// TIA Portal V16 export
// export: Created 2021-11-12T13:32:03.5567282Z, ExportSetting WithDefaults, DisplayName Totally Integrated Automation Portal, DisplayVersion V16 Update 3, DisplayName TIA Portal Version Control Interface, DisplayVersion V16 Update 2, DisplayName TIA Portal Openness, DisplayVersion V16 Update 3, DisplayName SINAMICS Startdrive Advanced, DisplayVersion V16 Update 5, DisplayName SINAMICS Startdrive G130, G150, S120, S150, SINAMICS MV, S210, DisplayVersion V16 Update 5, DisplayName SINAMICS Startdrive G110M, G120, G120C, G120D, G120P, G115D, DisplayVersion V16 Update 5, DisplayName STEP 7 Professional, DisplayVersion V16 Update 3, DisplayName STEP 7 Safety, DisplayVersion V16, DisplayName WinCC UA Professional, DisplayVersion V16 Update 3
DATA_BLOCK "STATUS_110"   // DB201
{ S7_Optimized_Access := 'TRUE' }
VERSION : 0.1
// stored: AutoNumber true, DBAccessibleFromOPCUA true, IsOnlyStoredInLoadMemory false, IsRetainMemResEnabled false, IsWriteProtectedInAS false, MemoryReserve 100
   VAR
      xxxxx___BinarySensors___xxxxx : Byte;
      GL01_BG01 : Bool;   // Proximitní senzor - Koncák pro referenci
      GL01_BG01R : Bool;   // Proximitní senzor - Zarážka nahoře
      GL01_BG01V : Bool;   // Proximitní senzor - Zarážka dole
      GL01_BG02 : Bool;   // Optický senzor - Přítomnost přířezu v pozici po vykulení
      GM01_BG01R : Bool;   // Indukční senzor - Výtah 1 dole
      GM01_BG01V : Bool;   // Indukční senzor - Výtah 1 nahoře
      GM01_BG02R : Bool;   // Indukční senzor - Výtah 2 dole
      GM01_BG02V : Bool;   // Indukční senzor - Výtah 2 nahoře
      GM01_BG03R : Bool;   // Indukční senzor - Výtah 3 dole
      GM01_BG03V : Bool;   // Indukční senzor - Výtah 3 nahoře
      GM01_BG04R : Bool;   // Indukční senzor - Výtah 4 dole
      GM01_BG04V : Bool;   // Indukční senzor - Výtah 4 nahoře
      GL01_BG03 : Bool;   // Optický senzor - Přířez na řetěze před výtahama
      GM01_BG01 : Bool;   // Optický senzor - Přířez na řetěze výtah 1
      GM01_BG02 : Bool;   // Optický senzor - Přířez na řetěze výtah 2
      GM01_BG03 : Bool;   // Optický senzor - Přířez na řetěze výtah 3
      GM01_BG04 : Bool;   // Optický senzor - Přířez na řetěze výtah 4
      GL01_BG04 : Bool;   // Přířez na řetěze za posledním výtahem
      GL01_BG5 : Bool;   // Enkodér na dopravníku
      xxxxx___BinaryOthers___xxxxx : Byte;
      UH31_FC01 : Bool;   // Servodrive TA01 is OK / Servoměnič TA01 je OK
      UC10_FC21 : Bool;   // 230V Part align OK
      UC12_FC01 : Bool;   // 400V Conveyor OK
      SF01_14 : Bool;   // Conveyor Remote
      SF01_24 : Bool;   // Conveyor Automat
      SF03_14 : Bool;   // Conveyor Start automat
      SF04_12 : Bool;   // Conveyor Stop
      SF05_14 : Bool;   // Conveyor Manual backward
      SF05_24 : Bool;   // Conveyor Manual forward
      SF06_14 : Bool;   // Conveyor lift 1 up
      SF06_24 : Bool;   // Conveyor lift 1 down
      SF07_14 : Bool;   // Conveyor lift 2 up
      SF07_24 : Bool;   // Conveyor lift 2 down
      SF08_14 : Bool;   // Conveyor lift 3 up
      SF08_24 : Bool;   // Conveyor lift 3 down
      SF09_14 : Bool;   // Conveyor lift 4 up
      SF09_24 : Bool;   // Conveyor lift 4 down
      SF10_14 : Bool;   // Conveyor aligning align
      SF10_24 : Bool;   // Conveyor aligning release
      SF11_14 : Bool;   // Conveyor Stopper up
      SF11_24 : Bool;   // Conveyor Stopper down
      xxxxx___Drives___xxxxx : Byte;
      GL01_MA02 : Struct   // Conveyour - motor / Dopravník - motor
         Main : "UDT_Status_main";
         Specific { S7_SetPoint := 'True'} : "UDT_Drive1_Status_specific";
         Error : "UDT_Error01";
      END_STRUCT;
      UC12_TA01 : Struct   // Conveyour - G120 / Dopravník - měnič G120
         Main { S7_SetPoint := 'True'} : "UDT_Status_main";
         Specific { S7_SetPoint := 'True'} : "UDT_SINAMICS_G120_Status_specific";
         Error { S7_SetPoint := 'True'} : "UDT_Error02";
      END_STRUCT;
      GL01_BG05 : Struct   // Conveyour - encoder / Dopravník - enkodér
         Main : "UDT_Status_main";
         Specific : "UDT_MCEncoder_Status_specific";
         Error : "UDT_Error01";
      END_STRUCT;
      UH31_TA01 : Struct   // Servodrive - FESTO / Řízení servomotoru - FESTO
         Main : "UDT_Status_main";
         Specific { S7_SetPoint := 'True'} : "UDT_FESTO_CMMT_Status_specific";
         Error { S7_SetPoint := 'True'} : "UDT_Error02";
      END_STRUCT;
      xxxxx___Others___xxxxx : Byte;
      ConvReadyLoad : Bool;   // Station is ready for material / Stanice je připravena na příjem kusů
      GL01_MA01_HomePos : Bool;   // FESTO servo home position
      PartCounter : Int;   // Number of parts in gripper
      xxxxx___Valves___xxxxx : Byte;
      GL01_MM01 : Struct   // Valve - stopping / Pneumatický válec - Zarážka pro vykulení
         Main : "UDT_Status_main";
         Specific : "UDT_Valve2WB_Status_specific";
         Error : "UDT_Error01";
      END_STRUCT;
      GM01_MM01 : Struct   // Valve - Lift 1 / Pneumatický válec - Zvedání přířezu - Výtah 1
         Main : "UDT_Status_main";
         Specific : "UDT_Valve2WB_Status_specific";
         Error : "UDT_Error01";
      END_STRUCT;
      GM01_MM02 : Struct   // Valve - Lift 2 / Pneumatický válec - Zvedání přířezu - Výtah 2
         Main : "UDT_Status_main";
         Specific : "UDT_Valve2WB_Status_specific";
         Error : "UDT_Error01";
      END_STRUCT;
      GM01_MM03 : Struct   // Valve - Lift 3 / Pneumatický válec - Zvedání přířezu - Výtah 3
         Main : "UDT_Status_main";
         Specific : "UDT_Valve2WB_Status_specific";
         Error : "UDT_Error01";
      END_STRUCT;
      GM01_MM04 : Struct   // Valve - Lift 4 / Pneumatický válec - Zvedání přířezu - Výtah 4
         Main : "UDT_Status_main";
         Specific : "UDT_Valve2WB_Status_specific";
         Error : "UDT_Error01";
      END_STRUCT;
      xxxxx__SenzorAlarms__xxxxx : Byte;
      GL01_MM01_Alarm : Struct   // Stopper - sensor discrepance / Diskrepance senzorů na pozici zarážky.
         Main { S7_SetPoint := 'True'} : "UDT_Status_main";
         Specific { S7_SetPoint := 'True'} : "UDT_DI_Mon_Status_specific";
         Error { S7_SetPoint := 'True'} : "UDT_Error01";
      END_STRUCT;
      GM01_MM01_Alarm : Struct   // Lift 1 - sensor discrepance / Diskrepance senzorů na pozici 1. výtahu.
         Main { S7_SetPoint := 'True'} : "UDT_Status_main";
         Specific { S7_SetPoint := 'True'} : "UDT_DI_Mon_Status_specific";
         Error { S7_SetPoint := 'True'} : "UDT_Error01";
      END_STRUCT;
      GM01_MM02_Alarm : Struct   // Lift 2 - sensor discrepance / Diskrepance senzorů na pozici 2. výtahu.
         Main { S7_SetPoint := 'True'} : "UDT_Status_main";
         Specific { S7_SetPoint := 'True'} : "UDT_DI_Mon_Status_specific";
         Error { S7_SetPoint := 'True'} : "UDT_Error01";
      END_STRUCT;
      GM01_MM03_Alarm : Struct   // Lift 3 - sensor discrepance / Diskrepance senzorů na pozici 3. výtahu.
         Main { S7_SetPoint := 'True'} : "UDT_Status_main";
         Specific { S7_SetPoint := 'True'} : "UDT_DI_Mon_Status_specific";
         Error { S7_SetPoint := 'True'} : "UDT_Error01";
      END_STRUCT;
      GM01_MM04_Alarm : Struct   // Lift 4 - sensor discrepance / Diskrepance senzorů na pozici 4. výtahu.
         Main { S7_SetPoint := 'True'} : "UDT_Status_main";
         Specific { S7_SetPoint := 'True'} : "UDT_DI_Mon_Status_specific";
         Error { S7_SetPoint := 'True'} : "UDT_Error01";
      END_STRUCT;
      xxxxx___ProcessAlarms___xxxxx : Byte;
      DataTracking_1 : Struct   // Part in stopping position not on map / Kus na pozici zarážky není na mapě.
         Main : "UDT_Status_main";
         Specific : "UDT_DI_Mon_Status_specific";
         Error { S7_SetPoint := 'True'} : "UDT_Error01";
      END_STRUCT;
      DataTracking_2 : Struct   // Part in lift 1 position not on map / Kus na pozici 1. výtahu není na mapě.
         Main : "UDT_Status_main";
         Specific : "UDT_DI_Mon_Status_specific";
         Error { S7_SetPoint := 'True'} : "UDT_Error01";
      END_STRUCT;
      DataTracking_3 : Struct   // Part in lift 2 position not on map / Kus na pozici 2. výtahu není na mapě.
         Main : "UDT_Status_main";
         Specific : "UDT_DI_Mon_Status_specific";
         Error { S7_SetPoint := 'True'} : "UDT_Error01";
      END_STRUCT;
      DataTracking_4 : Struct   // Part in lift 3 position not on map / Kus na pozici 3. výtahu není na mapě.
         Main : "UDT_Status_main";
         Specific : "UDT_DI_Mon_Status_specific";
         Error { S7_SetPoint := 'True'} : "UDT_Error01";
      END_STRUCT;
      DataTracking_5 : Struct   // Part in lift 4 position not on map / Kus na pozici 4. výtahu není na mapě.
         Main : "UDT_Status_main";
         Specific : "UDT_DI_Mon_Status_specific";
         Error { S7_SetPoint := 'True'} : "UDT_Error01";
      END_STRUCT;
      DataTracking_6 : Struct   // Part in before lifts position not on map / Kus na pozici před výtahami naní na mapě.
         Main : "UDT_Status_main";
         Specific : "UDT_DI_Mon_Status_specific";
         Error { S7_SetPoint := 'True'} : "UDT_Error01";
      END_STRUCT;
      Senzor_1 : Struct   // Part in stopping position not on senzor / Kus na pozici zarážky není na senzoru.
         Main : "UDT_Status_main";
         Specific : "UDT_DI_Mon_Status_specific";
         Error { S7_SetPoint := 'True'} : "UDT_Error01";
      END_STRUCT;
      Senzor_2 : Struct   // Part in lift 1 position not on senzor / Kus na pozici 1. výtahu není na senzoru.
         Main : "UDT_Status_main";
         Specific : "UDT_DI_Mon_Status_specific";
         Error { S7_SetPoint := 'True'} : "UDT_Error01";
      END_STRUCT;
      Senzor_3 : Struct   // Part in lift 2 position not on senzor / Kus na pozici 2. výtahu není na senzoru.
         Main : "UDT_Status_main";
         Specific : "UDT_DI_Mon_Status_specific";
         Error { S7_SetPoint := 'True'} : "UDT_Error01";
      END_STRUCT;
      Senzor_4 : Struct   // Part in lift 3 position not on senzor / Kus na pozici 3. výtahu není na senzoru.
         Main : "UDT_Status_main";
         Specific : "UDT_DI_Mon_Status_specific";
         Error { S7_SetPoint := 'True'} : "UDT_Error01";
      END_STRUCT;
      Senzor_5 : Struct   // Part in lift 4 position not on senzor / Kus na pozici 4. výtahu není na senzoru.
         Main : "UDT_Status_main";
         Specific : "UDT_DI_Mon_Status_specific";
         Error { S7_SetPoint := 'True'} : "UDT_Error01";
      END_STRUCT;
      Senzor_6 : Struct   // Part in before lifts position not on senzor / Kus na pozici před výtahami naní na senzoru.
         Main : "UDT_Status_main";
         Specific : "UDT_DI_Mon_Status_specific";
         Error { S7_SetPoint := 'True'} : "UDT_Error01";
      END_STRUCT;
      UC10_FC21_Alarm : Struct   // 230V Part align NOK / 230V zarovnávání kusů NOK
         Main { S7_SetPoint := 'True'} : "UDT_Status_main";
         Specific { S7_SetPoint := 'True'} : "UDT_DI_Mon_Status_specific";
         Error { S7_SetPoint := 'True'} : "UDT_Error01";
      END_STRUCT;
      UC12_FC01_Alarm : Struct   // 400V Conveyor NOK / 400V pohon dopravníku NOK
         Main { S7_SetPoint := 'True'} : "UDT_Status_main";
         Specific { S7_SetPoint := 'True'} : "UDT_DI_Mon_Status_specific";
         Error { S7_SetPoint := 'True'} : "UDT_Error01";
      END_STRUCT;
      ConvOverflow : Struct   // Part behind last lift / Kus za posledním výtahem.
         Main : "UDT_Status_main";
         Specific : "UDT_DI_Mon_Status_specific";
         Error { S7_SetPoint := 'True'} : "UDT_Error01";
      END_STRUCT;
      ConvStepTooLong : Struct   // Conveyor step is too long / Krok dopravníku je příliš dlouhý.
         Main : "UDT_Status_main";
         Specific : "UDT_DI_Mon_Status_specific";
         Error { S7_SetPoint := 'True'} : "UDT_Error01";
      END_STRUCT;
      xxxxx__MaterialFlow__xxxxx : Byte;
   END_VAR
   VAR RETAIN
      MatCard : Array[1..28, 1..1] of "UDT_MatCard";
   END_VAR
BEGIN
END_DATA_BLOCK
